Yaskawa INFORM job: KRIS3(-160_-90)54.JBI

/JOB
//NAME KRIS3(-160_-90)54
//POS
///NPOS 270,270,270,20,0,0
///TOOL 0
///POSTYPE PULSE
///PULSE
C00000=36470,-76528,-106815,-19279,71473,-77234
C00001=136908,-99459,-124829,-20670,71348,-76391
C00002=134470,-76528,-106815,-19279,71473,-77234
C00003=159578,-94739,-111578,-14965,102577,-71346
C00004=157566,-87256,-71357,-3912,80960,-68626
C00005=176880,-68125,-57902,-5422,83635,-62119
C00006=177907,-68461,-55745,-5507,82211,-61705
C00007=177907,-68063,-54493,-5513,81648,-61681
C00008=177907,-68139,-54730,-5512,81754,-61686
C00009=178677,-69433,-55362,-5571,81531,-61412
C00010=178017,-68613,-55721,-5516,82126,-61665
C00011=169648,-85474,-89038,-4887,93378,-64966
C00012=163611,-44630,-68122,-4506,101126,-67267
C00013=165231,-48362,-64740,-4579,97228,-66587
C00014=165334,-48746,-64513,-4584,96897,-66540
C00015=165334,-48893,-63576,-4578,96247,-66515
C00016=165334,-48879,-63681,-4579,96319,-66517
C00017=165646,-49837,-64080,-4605,96090,-66402
C00018=165334,-48746,-64513,-4584,96897,-66540
C00019=140979,-108094,-110643,-2385,93763,-74547
C00020=140979,-108094,-110643,-2385,93763,-74547
C00021=140979,-108094,-110643,-2385,93763,-74547
C00022=140979,-108094,-110643,-2385,93763,-74547
C00023=140979,-108246,-109289,-2383,92853,-74530
C00024=140979,-108231,-109453,-2383,92961,-74533
C00025=141280,-110659,-110301,-2409,92244,-74420
C00026=140979,-108094,-110643,-2385,93763,-74547
C00027=156700,-55897,-85418,8720,99373,-67438
C00028=156898,-58036,-83987,8629,97394,-67513
C00029=156898,-58722,-82817,8603,96332,-67586
C00030=156898,-58622,-82997,8608,96491,-67574
C00031=157341,-60416,-83948,8523,96115,-67457
C00032=156898,-58036,-83987,8629,97394,-67513
C00033=161369,-86849,-99090,-4273,98390,-67906
C00034=167909,-84037,-82934,3708,84523,-64877
C00035=168571,-85124,-82512,3609,83677,-64677
C00036=168571,-84898,-80901,3613,82804,-64704
C00037=168571,-84936,-81149,3613,82937,-64700
C00038=169203,-86467,-81802,3516,82525,-64499
C00039=168571,-85124,-82512,3609,83677,-64677
C00040=165600,-121955,-98284,4061,74695,-65975
C00041=174461,-109455,-70225,9835,59183,-64105
C00042=175080,-109402,-69148,9749,58483,-63930
C00043=175080,-108469,-67668,9792,58058,-63969
C00044=175080,-108628,-67921,9785,58130,-63962
C00045=176152,-109889,-68298,9565,57596,-63593
C00046=175080,-109402,-69148,9749,58483,-63930
C00047=145436,-132582,-96247,390,75065,-72870
C00048=145436,-132678,-96385,390,75101,-72870
C00049=145436,-153478,-122593,390,33069,-72870
C00050=145436,-153478,-122593,390,33069,-72870
C00051=145875,-137224,-99164,151,44123,-76557
C00052=145875,-137224,-99164,-3186,26783,-75636
C00053=145875,-137224,-99164,-3186,26783,-75636
C00054=126920,-141995,-100488,14842,27437,-88451
C00055=126921,-139435,-97257,15195,26791,-88624
C00056=126921,-140260,-98306,15082,27005,-88567
C00057=126657,-136107,-97292,14665,28515,-88375
C00058=126920,-141995,-100488,14842,27437,-88451
C00059=153689,-122615,-92358,7246,28662,-82796
C00060=153689,-122359,-91923,7277,28527,-82812
C00061=153689,-121251,-90046,7417,27945,-82882
C00062=153689,-121596,-90629,7373,28125,-82859
C00063=152562,-118169,-89603,8504,29355,-83484
C00064=153689,-122359,-91923,7277,28527,-82812
C00065=153734,-144670,-102026,-12528,26386,-79802
C00066=148920,-141423,-91163,-14854,15551,-80235
C00067=148967,-137496,-86916,-15534,14983,-79917
C00068=147891,-134819,-86332,-12174,15793,-81580
C00069=147123,-134668,-89168,-6588,20492,-83847
C00070=147184,-133728,-87772,-6813,20125,-83735
C00071=149705,-139389,-87494,-17948,14535,-78726
C00072=140769,-160579,-91179,-72763,19950,-46602
C00073=129302,-154781,-89703,-59410,13959,-54584
C00074=128993,-152913,-89439,-56337,14227,-56040
C00075=129214,-154274,-89633,-58559,14027,-54988
C00076=129214,-151990,-87339,-59384,13900,-54610
C00077=129539,-156129,-91089,-59119,14177,-54682
C00078=130002,-156587,-91482,-58522,14566,-54861
C00079=131612,-152018,-92345,-56188,18115,-55777
C00080=137260,-138866,-133764,-10166,31487,-76482
C00081=55962,-149633,-123442,-11923,14089,-75671
C00082=31464,-162597,-133764,-10166,12061,-76482
C00083=-11401,-148032,-125425,-11667,35640,-75771
C00084=-126225,-114648,-117375,-36487,17100,-65054
C00085=-160935,-140983,-109640,-13468,75088,-74332
C00086=-169853,-118963,-84593,-12681,69660,86771
C00087=-166041,-110678,-74459,-13320,68331,88303
C00088=-166223,-108797,-70951,-13405,67140,88373
C00089=-166223,-107663,-69097,-13458,66595,88438
C00090=-166223,-107867,-69431,-13449,66693,88427
C00091=-167322,-109580,-69957,-13369,65975,88109
C00092=-166243,-109210,-71582,-13386,67309,88347
C00093=-169217,-106350,-70409,-12947,67561,87233
C00094=-169217,-106256,-70250,-12951,67512,87238
C00095=-169217,-105112,-68312,-13006,66921,87306
C00096=-169217,-105283,-68599,-12998,67008,87297
C00097=-170397,-106999,-69102,-12897,66265,86949
C00098=-167930,-107758,-71144,-13135,67501,87709
C00099=-168330,-125239,-100831,-12460,76505,86600
C00100=-155830,-85289,-85709,-13656,89459,89593
C00101=-155617,-85922,-82565,-13677,87294,89905
C00102=-155617,-85683,-81004,-13681,86480,89993
C00103=-155617,-85728,-81276,-13680,86620,89979
C00104=-156391,-88450,-82422,-13606,85816,89798
C00105=-155763,-86416,-82528,-13661,87001,89886
C00106=-155923,-87175,-84120,-13644,87549,89771
C00107=-155609,-85916,-82709,-13676,87386,89897
C00108=-155609,-85729,-81437,-13679,86718,89971
C00109=-155609,-85763,-81652,-13678,86829,89960
C00110=-156185,-87803,-82513,-13623,86229,89826
C00111=-155614,-85958,-82864,-13674,87458,89888
C00112=-155923,-85281,-100905,-13881,98543,88548
C00113=-155518,-83496,-100141,-13947,99043,88626
C00114=-155147,-83263,-96119,-13888,96814,89004
C00115=-155147,-83507,-95337,-13865,96223,89071
C00116=-155147,-83457,-95507,-13869,96351,89056
C00117=-155768,-86094,-96638,-13778,95608,88929
C00118=-155255,-83510,-96958,-13888,97175,88925
C00119=-154682,-87233,-101845,693,104782,88208
C00120=-154005,-85079,-98247,676,103668,88429
C00121=-154005,-85354,-97445,675,103031,88426
C00122=-154005,-85287,-97652,675,103193,88426
C00123=-154486,-87439,-98578,683,102661,88260
C00124=-154216,-85718,-99521,682,104126,88361
C00125=-156826,-87943,-103938,737,105722,87490
C00126=-169505,-149944,-134809,912,70958,83129
C00127=-207316,-122712,-123448,7636,86368,80631
C00128=-224855,-108358,-71229,12006,64036,72649
C00129=-217077,-74631,-23766,41947,48629,49537
C00130=-218892,-67424,-12026,68960,50607,41965
C00131=-212692,-64398,-6060,71724,46143,41638
C00132=-212692,-63310,-4348,72177,45977,41343
C00133=-212692,-64398,-6060,71724,46143,41638
C00134=-210575,-63691,-5764,71905,44943,42037
C00135=-212692,-64398,-6060,71724,46143,41638
C00136=-222676,-51835,-4012,66283,54122,43011
C00137=-220683,-43055,3882,66739,52777,43150
C00138=-220683,-41728,6197,67257,52470,42760
C00139=-220683,-43055,3882,66739,52777,43150
C00140=-218176,-42178,4378,66898,51329,43628
C00141=-220683,-43055,3882,66739,52777,43150
C00142=-234013,-57846,-7460,65247,60464,40769
C00143=-233739,-55371,-8506,61318,66043,45868
C00144=-224021,-72963,-6178,68579,55797,42417
C00145=-222956,-69762,-1623,69618,54766,41957
C00146=-220957,-69447,-1516,70121,53696,42256
C00147=-222193,-69648,-1584,69812,54356,42072
C00148=-222502,-68090,774,70157,54288,41693
C00149=-222193,-69648,-1584,69812,54356,42072
C00150=-225636,-56152,5458,67261,57288,42948
C00151=-149006,-93113,-100988,5480,101691,74295
C00152=-149599,-96300,-103483,5484,101628,74092
C00153=-219127,-73013,-224,68618,57817,46460
C00154=-228607,-72912,-7621,63442,64869,47367
C00155=-220423,-75882,-15995,70402,50905,40654
C00156=-212092,-63463,-4317,72649,45688,41298
C00157=-163022,-96735,-99152,-22140,103253,76925
C00158=-162158,-93804,-96763,-22109,103515,77196
C00159=-220673,-36477,9481,67037,52832,43066
C00160=-225006,-42245,766,65045,56479,43585
C00161=-234485,-59648,-18556,62655,63569,43382
C00162=-203757,-97365,-58564,4219,60682,62576
C00163=-234472,-129171,-97928,9356,71113,51987
C00164=-234472,-150736,-135181,8964,82814,52858
C00165=-234472,-150736,-135181,8964,82814,52858
C00166=-215909,-75798,-109600,6127,103741,60188
C00167=-142211,-189130,-127292,69248,52498,52988
C00168=-118502,-172484,-110233,52609,25212,65150
C00169=-171509,-133648,-100111,8061,78079,67623
C00170=-179980,-112353,-73580,8533,73608,64392
C00171=-172896,-96696,-66298,2439,82915,67706
C00172=-163006,-94576,-83573,-21494,95359,78388
C00173=-162142,-91714,-81191,-21448,95589,78662
C00174=-161445,-106166,-69505,2991,79646,71488
C00175=-161519,-107811,-73451,2977,81228,71500
C00176=-162580,-105162,-72246,-8409,75537,72147
C00177=-166515,-102401,-68173,-8273,74056,70883
C00178=-163006,-94576,-83573,-21494,95359,78388
C00179=-162142,-91714,-81191,-21448,95589,78662
C00180=-175761,-93408,-64742,-7691,75635,67570
C00181=-169252,-115124,-101169,-7872,87423,69075
C00182=-154261,-79873,-81468,-8571,94879,73696
C00183=-155062,-80931,-79256,-8513,92911,73559
C00184=-163006,-94576,-83573,-21494,95359,78388
C00185=-162142,-91714,-81191,-21448,95589,78662
C00186=-163211,-72770,-75533,-8210,93956,70713
C00187=-163718,-69809,-76291,-8220,95872,70416
C00188=-152145,-81088,-82167,-2065,97703,74759
C00189=-153291,-82185,-80570,-2065,96129,74395
C00190=-163006,-94576,-83573,-21494,95359,78388
C00191=-162142,-91714,-81191,-21448,95589,78662
C00192=-143402,-88471,-83234,-1964,94787,77778
C00193=-144574,-84995,-103251,-2104,108854,77145
C00194=-151765,-102418,-106955,5657,95758,75438
C00195=-150608,-101637,-104194,5548,94387,75768
C00196=-163006,-94576,-83573,-21494,95359,78388
C00197=-162142,-91714,-81191,-21448,95589,78662
C00198=-139211,-109713,-107103,4584,91330,79466
C00199=-143989,-108966,-109417,5008,93413,77941
C00200=-143223,-109509,-108756,-8615,88663,77081
C00201=-143797,-107565,-105457,-8538,87583,76960
C00202=-163006,-94576,-83573,-21494,95359,78388
C00203=-162142,-91714,-81191,-21448,95589,78662
C00204=-154250,-98677,-102309,-7016,89198,73353
C00205=-144143,-146387,-128453,-8544,81812,77235
C00206=-130399,-165491,-128261,582,73715,81342
C00207=-149731,-158641,-113843,-14975,70738,-69794
C00208=-149731,-158641,-113843,-14975,70738,-69794
C00209=-126225,-114648,-117375,-36487,17100,-65054
C00210=-118781,-153853,-134406,-32592,23357,-65054
C00211=-12470,-167083,-125425,-11667,16324,-75771
C00212=137258,-84249,-120477,-10166,64820,-76482
C00213=160540,-100857,-113063,-23155,68829,-67581
C00214=182830,-114405,-112845,-16003,91175,-61677
C00215=183790,-123536,-112279,-16086,86512,-60735
C00216=173929,-95305,-100930,-8088,100256,-64859
C00217=158743,-95268,-103371,-5812,102972,-69826
C00218=157888,-92366,-100981,-5813,102933,-70115
C00219=164971,-109182,-106036,-7793,95435,-67600
C00220=164197,-113877,-111682,-7800,96401,-67923
C00221=173870,-143306,-120553,-7913,87764,-64082
C00222=171816,-118751,-98057,-3590,91441,-64891
C00223=176035,-116344,-93182,-3358,89860,-63416
C00224=158755,-94787,-86481,976,103949,-69303
C00225=157900,-91912,-84097,841,103969,-69603
C00226=165474,-127613,-96498,-3911,85645,-66872
C00227=163756,-130674,-100363,-3993,86365,-67475
C00228=177254,-154866,-106204,-3341,78153,-62695
C00229=194740,-128784,-79093,-2289,75465,-56815
C00230=199705,-123555,-74669,-1955,75552,-55172
C00231=158782,-86330,-62292,-2348,97119,-70521
C00232=157926,-83586,-59872,-2521,97014,-70811
C00233=188878,-135549,-77220,-2730,70669,-58654
C00234=186334,-138981,-80518,-2891,70851,-59497
C00235=202790,-114657,-73561,7469,64730,-55511
C00236=205310,-109506,-69417,7096,64604,-54603
C00237=158743,-95268,-103371,-5812,102972,-69826
C00238=157888,-92366,-100981,-5813,102933,-70115
C00239=208506,-101173,-65845,8459,63334,-53705
C00240=188075,-151957,-103997,12598,63075,-61358
C00241=175676,-115929,-94468,13375,77380,-64283
C00242=179228,-108031,-88427,12897,77138,-63049
C00243=158755,-94787,-86481,976,103949,-69303
C00244=157900,-91912,-84097,841,103969,-69603
C00245=187549,-93923,-83081,11553,79750,-59861
C00246=178297,-108275,-107099,12771,88378,-62209
C00247=165278,-79866,-95804,14582,97947,-65562
C00248=167332,-81697,-93226,14245,95145,-65199
C00249=158782,-86330,-62292,-2348,97119,-70521
C00250=157926,-83586,-59872,-2521,97014,-70811
C00251=172083,-74876,-89232,15991,93470,-63478
C00252=166883,-83368,-97274,16810,95013,-65031
C00253=148381,-154133,-120540,18986,77988,-74048
C00254=148381,-154133,-120540,18986,29025,-74048
C00255=148381,-154133,-120540,18986,29025,-74048
C00256=148381,-154133,-120540,18986,29025,-74048
C00257=148381,-154133,-120540,635,27393,-68347
C00258=131809,-160671,-109428,31686,20564,-84507
C00259=131822,-150122,-103532,29341,22114,-83385
C00260=161827,-137088,-100610,-19196,25445,-57865
C00261=160079,-162229,-113551,-20584,20355,-57319
C00262=127848,-170739,-113822,-25929,20694,-59837
C00263=98584,-145628,-105124,27441,32859,-85558
C00264=101235,-136742,-99408,24366,32991,-83733
C00265=148832,-132035,-98353,-25409,35327,-54782
C00266=162526,-150393,-107796,-38053,37342,-46820
C00267=161637,-148332,-107324,-36893,37578,-47548
C00268=136473,-81821,-106853,-20577,68974,-75046
C00269=36470,-76528,-106815,-19279,71473,-77234
BC00000=293716,514317,1072451
BC00001=351926,331601,1072451
BC00002=351926,292903,1072451
BC00003=351926,213013,1072451
BC00004=381341,211891,1072451
BC00005=381341,211891,1072451
BC00006=381341,211891,1072451
BC00007=381341,211891,1072451
BC00008=381341,211891,1072451
BC00009=381341,211891,1072451
BC00010=381341,211891,1072451
BC00011=381341,211891,1072448
BC00012=381341,211891,1072448
BC00013=381341,211891,1072448
BC00014=381341,211891,1072448
BC00015=381341,211891,1072448
BC00016=381341,211891,1072448
BC00017=381341,211891,1072448
BC00018=381341,211891,1072448
BC00019=327940,182383,1072451
BC00020=327940,158933,1072451
BC00021=323570,159157,1054517
BC00022=322810,158773,1051038
BC00023=322810,158773,1051038
BC00024=322810,158773,1051038
BC00025=322810,158773,1051038
BC00026=322810,158773,1051038
BC00027=324758,182517,1072451
BC00028=324758,182517,1072451
BC00029=324758,182517,1072451
BC00030=324758,182517,1072451
BC00031=324758,182517,1072451
BC00032=324758,182517,1072451
BC00033=323103,182517,1072451
BC00034=323103,182517,1072451
BC00035=323103,182517,1072451
BC00036=323103,182517,1072451
BC00037=323103,182517,1072451
BC00038=323103,182517,1072451
BC00039=323103,182517,1072451
BC00040=323103,182517,1072451
BC00041=323103,182517,1072451
BC00042=323103,182517,1072451
BC00043=323103,182517,1072451
BC00044=323103,182517,1072451
BC00045=323103,182517,1072451
BC00046=323103,182517,1072451
BC00047=332426,182517,1072451
BC00048=332426,182517,1072451
BC00049=332426,227917,1072451
BC00050=367924,391941,1072451
BC00051=367924,391941,1072451
BC00052=323298,308265,712615
BC00053=297724,284937,708891
BC00054=297724,284937,708891
BC00055=297724,284937,708889
BC00056=297724,284937,708889
BC00057=297724,284937,708889
BC00058=297724,284937,708891
BC00059=297724,284937,708891
BC00060=297724,284937,708891
BC00061=297724,284937,708891
BC00062=297724,284937,708891
BC00063=297724,284937,708891
BC00064=297724,284937,708891
BC00065=325419,295206,714526
BC00066=325419,295206,704236
BC00067=325419,295206,704234
BC00068=325419,295206,704234
BC00069=325419,295206,704234
BC00070=325419,295206,704234
BC00071=325419,295206,704234
BC00072=319446,285786,704234
BC00073=319446,285786,704234
BC00074=319446,285786,704234
BC00075=319446,285786,704234
BC00076=319446,285786,704234
BC00077=319446,285786,704234
BC00078=306058,333731,968548
BC00079=310610,415570,1064706
BC00080=352207,264891,1072451
BC00081=372153,109357,1072451
BC00082=378164,62489,1072451
BC00083=396581,158595,1072451
BC00084=311023,50823,1072451
BC00085=339144,73580,1072451
BC00086=339157,74032,1072451
BC00087=339157,74032,1072451
BC00088=339157,74032,1072451
BC00089=339157,74032,1072451
BC00090=339157,74032,1072451
BC00091=339157,74032,1072451
BC00092=339157,74032,1072451
BC00093=372221,74032,1072451
BC00094=372221,74032,1072451
BC00095=372221,74032,1072451
BC00096=372221,74032,1072451
BC00097=372221,74032,1072451
BC00098=372221,74032,1072451
BC00099=372221,74032,1072451
BC00100=372221,74032,1072451
BC00101=372221,74032,1072451
BC00102=372221,74032,1072451
BC00103=372221,74032,1072451
BC00104=372221,74032,1072451
BC00105=372221,74032,1072451
BC00106=338445,74032,1072451
BC00107=338445,73232,1069168
BC00108=338445,73232,1069168
BC00109=338445,73232,1069168
BC00110=338445,73232,1069168
BC00111=338445,73232,1069168
BC00112=338445,73232,1071030
BC00113=338445,99622,1071030
BC00114=338445,99622,1071030
BC00115=338445,99622,1071030
BC00116=338445,99622,1071030
BC00117=338445,99622,1071030
BC00118=338445,99622,1071030
BC00119=338445,99622,1071030
BC00120=338445,99622,1071030
BC00121=338445,99622,1071030
BC00122=338445,99622,1071030
BC00123=338445,99622,1071030
BC00124=338445,99622,1071030
BC00125=338445,99622,1071030
BC00126=338445,99622,1071030
BC00127=395065,437,1069903
BC00128=395065,437,1069903
BC00129=395065,437,1069903
BC00130=395065,437,1069903
BC00131=395065,437,1069903
BC00132=395065,437,1069903
BC00133=395065,437,1069903
BC00134=395065,437,1069903
BC00135=395065,437,1069903
BC00136=395065,437,1069903
BC00137=395065,437,1069903
BC00138=395065,437,1069903
BC00139=395065,437,1069903
BC00140=395065,437,1069903
BC00141=395065,437,1069903
BC00142=395065,437,1069903
BC00143=395064,1123,1069901
BC00144=395064,1123,1069901
BC00145=395064,1123,1069901
BC00146=395064,1123,1069901
BC00147=395064,1123,1069901
BC00148=395064,1123,1069901
BC00149=395064,1123,1069901
BC00150=395064,1123,1069901
BC00151=347303,98646,1072451
BC00152=347303,98646,1072451
BC00153=395064,1123,1069901
BC00154=395064,1123,1069901
BC00155=395064,1123,1069901
BC00156=395064,1123,1069901
BC00157=320927,137430,1072451
BC00158=320927,137430,1072451
BC00159=395064,1123,1069901
BC00160=395064,1123,1069901
BC00161=395064,1123,1069901
BC00162=395064,1123,1069901
BC00163=395064,22229,1069901
BC00164=395064,22229,1069901
BC00165=395064,111405,1069901
BC00166=395064,111405,1069901
BC00167=307195,19114,1039924
BC00168=312628,21569,1045452
BC00169=339157,74031,1072445
BC00170=339157,74031,1072445
BC00171=339157,74031,1072445
BC00172=320853,110629,1072451
BC00173=320853,110629,1072451
BC00174=339157,74031,1072445
BC00175=339157,74031,1072445
BC00176=339157,74031,1072445
BC00177=339157,74031,1072445
BC00178=320853,110629,1072451
BC00179=320853,110629,1072451
BC00180=339157,74031,1072445
BC00181=339157,74031,1072445
BC00182=339157,74031,1072445
BC00183=339157,74031,1072445
BC00184=320853,110629,1072451
BC00185=320853,110629,1072451
BC00186=339157,74031,1072445
BC00187=339157,74031,1072445
BC00188=339157,74031,1072445
BC00189=339157,74031,1072445
BC00190=320853,110629,1072451
BC00191=320853,110629,1072451
BC00192=339157,74031,1072445
BC00193=339157,74031,1072445
BC00194=321867,96463,1067741
BC00195=321867,96463,1067741
BC00196=320853,110629,1072451
BC00197=320853,110629,1072451
BC00198=321867,96463,1067741
BC00199=321867,96463,1067741
BC00200=321867,96463,1067741
BC00201=321867,96463,1067741
BC00202=320853,110629,1072451
BC00203=320853,110629,1072451
BC00204=321867,96463,1067741
BC00205=321867,96463,1067741
BC00206=331832,83535,1070452
BC00207=339144,73580,1072451
BC00208=339144,73580,1072451
BC00209=311023,50823,1072451
BC00210=311023,50823,1072451
BC00211=396581,158595,1072451
BC00212=352208,264890,1072451
BC00213=380287,222292,1072451
BC00214=345793,144315,1072448
BC00215=345793,144315,1072448
BC00216=345793,144315,1072448
BC00217=363046,147874,1072451
BC00218=363046,147874,1072451
BC00219=345793,144315,1072448
BC00220=346013,144317,1072448
BC00221=346013,144317,1072448
BC00222=336959,144429,1072450
BC00223=336960,144428,1072447
BC00224=363165,149824,1072451
BC00225=363165,149824,1072451
BC00226=336960,144428,1072447
BC00227=336960,144428,1072447
BC00228=336960,144428,1072447
BC00229=336960,144428,1072447
BC00230=336960,144428,1072447
BC00231=353911,176435,1072451
BC00232=353911,176435,1072451
BC00233=336960,144428,1072447
BC00234=336960,144428,1072447
BC00235=336960,144428,1072447
BC00236=336960,144428,1072447
BC00237=363046,147874,1072451
BC00238=363046,147874,1072451
BC00239=336960,144428,1072447
BC00240=336960,144428,1072447
BC00241=336960,144428,1072447
BC00242=336960,144428,1072447
BC00243=363165,149824,1072451
BC00244=363165,149824,1072451
BC00245=336960,144428,1072447
BC00246=336960,144428,1072447
BC00247=336960,144428,1072447
BC00248=336960,144428,1072447
BC00249=353911,176435,1072451
BC00250=353911,176435,1072451
BC00251=336960,144428,1072447
BC00252=336960,144428,1072447
BC00253=336960,144428,1072447
BC00254=376956,227130,1072447
BC00255=384452,390236,1072447
BC00256=384452,390236,786592
BC00257=345962,304340,657091
BC00258=316411,279825,657091
BC00259=316411,279825,657091
BC00260=299501,279825,657091
BC00261=316411,279825,657091
BC00262=329749,298472,657091
BC00263=315017,300783,657091
BC00264=315017,300783,657091
BC00265=312927,300783,657091
BC00266=315017,300783,657091
BC00267=315017,430587,912822
BC00268=349205,500385,1060684
BC00269=293716,514317,1072451
EC00000=1418945,372643
EC00001=1418945,372643
EC00002=1418945,372643
EC00003=1418945,372643
EC00004=1418945,372643
EC00005=1418945,372643
EC00006=1418945,372643
EC00007=1418945,372643
EC00008=1418945,372643
EC00009=1418945,372643
EC00010=1418945,372643
EC00011=1418944,372643
EC00012=1418944,372643
EC00013=1418944,372643
EC00014=1418944,372643
EC00015=1418944,372643
EC00016=1418944,372643
EC00017=1418944,372643
EC00018=1418944,372643
EC00019=1418945,372643
EC00020=1418945,372643
EC00021=1418945,372643
EC00022=1418945,372643
EC00023=1418945,372643
EC00024=1418945,372643
EC00025=1418945,372643
EC00026=1418945,372643
EC00027=1418945,372643
EC00028=1418945,372643
EC00029=1418945,372643
EC00030=1418945,372643
EC00031=1418945,372643
EC00032=1418945,372643
EC00033=1418945,372643
EC00034=1418945,372643
EC00035=1418945,372643
EC00036=1418945,372643
EC00037=1418945,372643
EC00038=1418945,372643
EC00039=1418945,372643
EC00040=1418945,372643
EC00041=1418945,372643
EC00042=1418945,372643
EC00043=1418945,372643
EC00044=1418945,372643
EC00045=1418945,372643
EC00046=1418945,372643
EC00047=1418945,372643
EC00048=1418945,372643
EC00049=1418945,372643
EC00050=1418945,372643
EC00051=1418945,372643
EC00052=1418945,372643
EC00053=1418945,372643
EC00054=1418945,372643
EC00055=1418944,372643
EC00056=1418944,372643
EC00057=1418944,372643
EC00058=1418945,372643
EC00059=1418945,372643
EC00060=1418945,372643
EC00061=1418945,372643
EC00062=1418945,372643
EC00063=1418945,372643
EC00064=1418945,372643
EC00065=1418945,372643
EC00066=1418945,372643
EC00067=1418945,372643
EC00068=1418945,372643
EC00069=1418945,372643
EC00070=1418945,372643
EC00071=1418945,372643
EC00072=1418945,372643
EC00073=1418945,372643
EC00074=1418945,372643
EC00075=1418945,372643
EC00076=1418945,372643
EC00077=1418945,372643
EC00078=1418945,372643
EC00079=1418945,372643
EC00080=1418945,372643
EC00081=1418945,372643
EC00082=1418945,372643
EC00083=1595090,-179995
EC00084=1773681,-740307
EC00085=1773681,-740307
EC00086=1773681,-740307
EC00087=1773681,-740307
EC00088=1773681,-740307
EC00089=1773681,-740307
EC00090=1773681,-740307
EC00091=1773681,-740307
EC00092=1773681,-740307
EC00093=1773681,-740307
EC00094=1773681,-740307
EC00095=1773681,-740307
EC00096=1773681,-740307
EC00097=1773681,-740307
EC00098=1773681,-740307
EC00099=1773681,-740307
EC00100=1773681,-740307
EC00101=1773681,-740307
EC00102=1773681,-740307
EC00103=1773681,-740307
EC00104=1773681,-740307
EC00105=1773681,-740307
EC00106=1773681,-740307
EC00107=1773681,-740307
EC00108=1773681,-740307
EC00109=1773681,-740307
EC00110=1773681,-740307
EC00111=1773681,-740307
EC00112=1773681,-740307
EC00113=1773681,-740307
EC00114=1773681,-740307
EC00115=1773681,-740307
EC00116=1773681,-740307
EC00117=1773681,-740307
EC00118=1773681,-740307
EC00119=1773681,-740307
EC00120=1773681,-740307
EC00121=1773681,-740307
EC00122=1773681,-740307
EC00123=1773681,-740307
EC00124=1773681,-740307
EC00125=1773681,-740307
EC00126=1773681,-740307
EC00127=1773681,-740307
EC00128=1773681,-740307
EC00129=1773681,-740307
EC00130=1773681,-740307
EC00131=1773681,-740307
EC00132=1773681,-740307
EC00133=1773681,-740307
EC00134=1773681,-740307
EC00135=1773681,-740307
EC00136=1773681,-740307
EC00137=1773681,-740307
EC00138=1773681,-740307
EC00139=1773681,-740307
EC00140=1773681,-740307
EC00141=1773681,-740307
EC00142=1773681,-740307
EC00143=1773685,-740307
EC00144=1773685,-740307
EC00145=1773685,-740307
EC00146=1773685,-740307
EC00147=1773685,-740307
EC00148=1773685,-740307
EC00149=1773685,-740307
EC00150=1773685,-740307
EC00151=1773681,-740307
EC00152=1773681,-740307
EC00153=1773685,-740307
EC00154=1773685,-740307
EC00155=1773685,-740307
EC00156=1773685,-740307
EC00157=1773681,-740307
EC00158=1773681,-740307
EC00159=1773685,-740307
EC00160=1773685,-740307
EC00161=1773685,-740307
EC00162=1773685,-740307
EC00163=1773685,-740307
EC00164=1773685,-740307
EC00165=1773685,-740307
EC00166=1773685,-740307
EC00167=1773681,-740307
EC00168=1773681,-740307
EC00169=1773683,-740305
EC00170=1773683,-740305
EC00171=1773683,-740305
EC00172=1773681,-740307
EC00173=1773681,-740307
EC00174=1773683,-740305
EC00175=1773683,-740305
EC00176=1773683,-740305
EC00177=1773683,-740305
EC00178=1773681,-740307
EC00179=1773681,-740307
EC00180=1773683,-740305
EC00181=1773683,-740305
EC00182=1773683,-740305
EC00183=1773683,-740305
EC00184=1773681,-740307
EC00185=1773681,-740307
EC00186=1773683,-740305
EC00187=1773683,-740305
EC00188=1773683,-740305
EC00189=1773683,-740305
EC00190=1773681,-740307
EC00191=1773681,-740307
EC00192=1773683,-740305
EC00193=1773683,-740305
EC00194=1773683,-740305
EC00195=1773683,-740305
EC00196=1773681,-740307
EC00197=1773681,-740307
EC00198=1773683,-740305
EC00199=1773683,-740305
EC00200=1773683,-740305
EC00201=1773683,-740305
EC00202=1773681,-740307
EC00203=1773681,-740307
EC00204=1773683,-740305
EC00205=1773683,-740305
EC00206=1773683,-740305
EC00207=1773681,-740307
EC00208=1773681,-740307
EC00209=1773681,-740307
EC00210=1773681,-740307
EC00211=1595090,-179995
EC00212=1418947,372636
EC00213=1418945,372643
EC00214=1418944,372643
EC00215=1418944,372643
EC00216=1418944,372643
EC00217=1418945,372643
EC00218=1418945,372643
EC00219=1418944,372643
EC00220=1418944,372643
EC00221=1418944,372643
EC00222=1418945,372643
EC00223=1418944,372643
EC00224=1418945,372643
EC00225=1418945,372643
EC00226=1418944,372643
EC00227=1418944,372643
EC00228=1418944,372643
EC00229=1418944,372643
EC00230=1418944,372643
EC00231=1418945,372643
EC00232=1418945,372643
EC00233=1418944,372643
EC00234=1418944,372643
EC00235=1418944,372643
EC00236=1418944,372643
EC00237=1418945,372643
EC00238=1418945,372643
EC00239=1418944,372643
EC00240=1418944,372643
EC00241=1418944,372643
EC00242=1418944,372643
EC00243=1418945,372643
EC00244=1418945,372643
EC00245=1418944,372643
EC00246=1418944,372643
EC00247=1418944,372643
EC00248=1418944,372643
EC00249=1418945,372643
EC00250=1418945,372643
EC00251=1418944,372643
EC00252=1418944,372643
EC00253=1418944,372643
EC00254=1418944,372643
EC00255=1418944,372643
EC00256=1418944,372643
EC00257=1418944,372643
EC00258=1418944,372643
EC00259=1418944,372643
EC00260=1418944,372643
EC00261=1418944,372643
EC00262=1418944,372643
EC00263=1418944,372643
EC00264=1418944,372643
EC00265=1418944,372643
EC00266=1418944,372643
EC00267=1418944,372643
EC00268=1418945,372643
EC00269=1418945,372643
///POSTYPE BASE
///RECTAN
///RCONF 0,0,0,0,1,0,0,0,0,0,0,0,0,0,0,0,0,0,0,0,0,0,0,0
P00006=2.006,1.622,-0.565,0.0000,0.0000,0.0000
P00021=0.073,2.058,-0.109,0.0000,0.0000,0.0000
P00022=2.006,1.622,-0.565,0.0000,0.0000,0.0000
///RCONF 0,0,0,0,0,0,0,0,0,0,0,0,0,0,0,0,0,0,0,0,0,0,0,0
P00023=-2.957,-4.083,2.762,0.0000,0.0000,0.0000
P00024=-1.466,-0.226,-0.419,0.0000,0.0000,0.0000
P00025=3.643,0.007,-2.585,0.0000,0.0000,0.0000
P00026=2.644,0.055,-2.583,0.0000,0.0000,0.0000
P00027=2.278,0.099,-4.210,0.0000,0.0000,0.0000
P00028=-1.778,-0.182,-2.050,0.0000,0.0000,0.0000
P00029=1.749,4.006,-0.261,0.0000,0.0000,0.0000
P00030=-0.014,-0.768,0.131,0.0000,0.0000,0.0000
P00031=-0.170,0.039,-0.647,0.0000,0.0000,0.0000
P00032=-0.423,0.157,3.222,0.0000,0.0000,0.0000
P00033=0.854,-1.099,3.047,0.0000,0.0000,0.0000
///RCONF 0,0,0,0,1,0,0,0,0,0,0,0,0,0,0,0,0,0,0,0,0,0,0,0
P00034=-8.151,9.743,-4.393,0.0000,0.0000,0.0000
///RCONF 0,0,0,0,0,0,0,0,0,0,0,0,0,0,0,0,0,0,0,0,0,0,0,0
P00035=0.390,-0.027,1.040,0.0000,0.0000,0.0000
P00036=-2.434,0.084,0.197,0.0000,0.0000,0.0000
P00037=-1.075,5.090,-3.949,0.0000,0.0000,0.0000
P00038=0.174,-1.527,-10.860,0.0000,0.0000,0.0000
P00039=-0.109,1.838,-0.266,0.0000,0.0000,0.0000
//INST
///DATE 2024/11/25 20:44
///ATTR SC,RW
///GROUP1 RB1,BS1
///GROUP2 ST1
NOP
MOVJ C00000 BC00000 VJ=100.00  +MOVJ EC00000 VJ=100.00
'MUZYLO 260124 START
MOVJ C00001 BC00001 VJ=100.00  +MOVJ EC00001 VJ=100.00
MOVJ C00002 BC00002 VJ=100.00  +MOVJ EC00002 VJ=100.00
MOVJ C00003 BC00003 VJ=100.00  +MOVJ EC00003 VJ=100.00
'Path S1422
SFTOF3D
MOVJ C00004 BC00004 VJ=100.00  +MOVJ EC00004 VJ=100.00
MOVL C00005 BC00005 V=400.0  +MOVJ EC00005 VJ=100.00
SMOVL C00006 BC00006 V=100.0  +MOVJ EC00006
SREFP 3 C00007 BC00007  +REFP EC00007
CALL JOB:SEARCH-R1-S13D
SET P021 P006
SFTON3D P021
SMOVL C00008 BC00008 V=100.0  +MOVJ EC00008
SREFP 3 C00009 BC00009  +REFP EC00009
CALL JOB:SEARCH-R1-S13D
SET P021 P006
SFTON3D P021
SMOVL C00010 BC00010 V=100.0  +MOVJ EC00010
MOVL C00011 BC00011 V=400.0  +MOVJ EC00011 VJ=100.00
MOVL C00012 BC00012 V=1000.0  +MOVJ EC00012 VJ=100.00
MOVJ C00013 BC00013 VJ=100.00  +MOVJ EC00013 VJ=100.00
'Path S1423
SFTOF3D
SMOVL C00014 BC00014 V=100.0  +MOVJ EC00014
SREFP 3 C00015 BC00015  +REFP EC00015
CALL JOB:SEARCH-R1-S13D
SET P022 P006
SFTON3D P022
SMOVL C00016 BC00016 V=100.0  +MOVJ EC00016
SREFP 3 C00017 BC00017  +REFP EC00017
CALL JOB:SEARCH-R1-S13D
SET P022 P006
SFTON3D P022
SMOVL C00018 BC00018 V=100.0  +MOVJ EC00018
MOVL C00019 BC00019 V=400.0  +MOVJ EC00019 VJ=100.00
MOVL C00020 BC00020 V=1000.0  +MOVJ EC00020 VJ=100.00
MOVJ C00021 BC00021 VJ=100.00  +MOVJ EC00021 VJ=100.00
'Path S1424
SFTOF3D
SMOVL C00022 BC00022 V=100.0  +MOVJ EC00022
SREFP 3 C00023 BC00023  +REFP EC00023
CALL JOB:SEARCH-R1-S13D
SET P023 P006
SFTON3D P023
SMOVL C00024 BC00024 V=100.0  +MOVJ EC00024
SREFP 3 C00025 BC00025  +REFP EC00025
CALL JOB:SEARCH-R1-S13D
SET P023 P006
SFTON3D P023
SMOVL C00026 BC00026 V=100.0  +MOVJ EC00026
MOVL C00027 BC00027 V=400.0  +MOVJ EC00027 VJ=100.00
SMOVL C00028 BC00028 V=100.0  +MOVJ EC00028
SREFP 3 C00029 BC00029  +REFP EC00029
CALL JOB:SEARCH-R1-S13D
SET P024 P006
SFTON3D P024
SMOVL C00030 BC00030 V=100.0  +MOVJ EC00030
SREFP 3 C00031 BC00031  +REFP EC00031
CALL JOB:SEARCH-R1-S13D
SET P024 P006
SFTON3D P024
SMOVL C00032 BC00032 V=100.0  +MOVJ EC00032
MOVL C00033 BC00033 V=400.0  +MOVJ EC00033 VJ=100.00
MOVL C00034 BC00034 V=1000.0  +MOVJ EC00034 VJ=100.00
'Path S1423
SFTOF3D
SMOVL C00035 BC00035 V=100.0  +MOVJ EC00035
SREFP 3 C00036 BC00036  +REFP EC00036
CALL JOB:SEARCH-R1-S13D
SET P025 P006
SFTON3D P025
SMOVL C00037 BC00037 V=100.0  +MOVJ EC00037
SREFP 3 C00038 BC00038  +REFP EC00038
CALL JOB:SEARCH-R1-S13D
SET P025 P006
SFTON3D P025
SMOVL C00039 BC00039 V=100.0  +MOVJ EC00039
MOVL C00040 BC00040 V=400.0  +MOVJ EC00040 VJ=100.00
MOVL C00041 BC00041 V=1000.0  +MOVJ EC00041 VJ=100.00
'Path S1424
SFTOF3D
SMOVL C00042 BC00042 V=100.0  +MOVJ EC00042
SREFP 3 C00043 BC00043  +REFP EC00043
CALL JOB:SEARCH-R1-S13D
SET P026 P006
SFTON3D P026
SMOVL C00044 BC00044 V=100.0  +MOVJ EC00044
SREFP 3 C00045 BC00045  +REFP EC00045
CALL JOB:SEARCH-R1-S13D
SET P026 P006
SFTON3D P026
SMOVL C00046 BC00046 V=100.0  +MOVJ EC00046
MOVL C00047 BC00047 V=400.0  +MOVJ EC00047 VJ=100.00
MOVJ C00048 BC00048 VJ=50.00  +MOVJ EC00048 VJ=50.00
MOVJ C00049 BC00049 VJ=100.00  +MOVJ EC00049 VJ=50.00
MOVJ C00050 BC00050 VJ=100.00  +MOVJ EC00050 VJ=50.00
MOVJ C00051 BC00051 VJ=100.00  +MOVJ EC00051 VJ=50.00
MOVJ C00052 BC00052 VJ=100.00  +MOVJ EC00052 VJ=50.00
MOVJ C00053 BC00053 VJ=100.00  +MOVJ EC00053 VJ=50.00
SFTOF3D
SMOVL C00054 BC00054 V=166.7  +MOVJ EC00054
SREFP 3 C00055 BC00055  +REFP EC00055
CALL JOB:SEARCH-R1-S13D
SET P027 P006
SFTON3D P027
SMOVL C00056 BC00056 V=100.0  +MOVJ EC00056
SREFP 3 C00057 BC00057  +REFP EC00057
CALL JOB:SEARCH-R1-S13D
SET P027 P006
SFTON3D P027
SMOVL C00058 BC00058 V=100.0  +MOVJ EC00058
SMOVL C00059 BC00059 V=416.7  +MOVJ EC00059
SFTOF3D
SMOVL C00060 BC00060 V=100.0  +MOVJ EC00060
SREFP 3 C00061 BC00061  +REFP EC00061
CALL JOB:SEARCH-R1-S13D
SET P028 P006
SFTON3D P028
SMOVL C00062 BC00062 V=100.0  +MOVJ EC00062
SREFP 3 C00063 BC00063  +REFP EC00063
CALL JOB:SEARCH-R1-S13D
SET P028 P006
SFTON3D P028
SMOVL C00064 BC00064 V=100.0  +MOVJ EC00064
SMOVL C00065 BC00065 V=416.7  +MOVJ EC00065
SMOVL C00066 BC00066 V=416.7  +MOVJ EC00066
SFTOF3D
SMOVL C00067 BC00067 V=100.0  +MOVJ EC00067
SREFP 3 C00068 BC00068  +REFP EC00068
CALL JOB:SEARCH-R1-S13D
SET P029 P006
SFTON3D P029
SMOVL C00069 BC00069 V=100.0  +MOVJ EC00069
SREFP 3 C00070 BC00070  +REFP EC00070
CALL JOB:SEARCH-R1-S13D
SET P029 P006
SFTON3D P029
SMOVL C00071 BC00071 V=100.0  +MOVJ EC00071
MOVJ C00072 BC00072 VJ=100.00  +MOVJ EC00072 VJ=50.00
SFTOF3D
SMOVL C00073 BC00073 V=83.3  +MOVJ EC00073
SREFP 3 C00074 BC00074  +REFP EC00074
CALL JOB:SEARCH-R1-S13D
SET P030 P006
SFTON3D P030
SMOVL C00075 BC00075 V=100.0  +MOVJ EC00075
SREFP 3 C00076 BC00076  +REFP EC00076
CALL JOB:SEARCH-R1-S13D
SET P030 P006
SFTON3D P030
SMOVL C00077 BC00077 V=100.0  +MOVJ EC00077
SFTOF3D
MOVL C00078 BC00078 V=1000.0  +MOVJ EC00078 VJ=100.00
'obrot
MOVJ C00079 BC00079 VJ=100.00  +MOVJ EC00079 VJ=100.00
MOVJ C00080 BC00080 VJ=100.00  +MOVJ EC00080 VJ=100.00
MOVJ C00081 BC00081 VJ=60.00  +MOVJ EC00081 VJ=15.00
MOVJ C00082 BC00082 VJ=100.00  +MOVJ EC00082 VJ=100.00
MOVJ C00083 BC00083 VJ=100.00  +MOVJ EC00083 VJ=100.00
MOVJ C00084 BC00084 VJ=100.00  +MOVJ EC00084 VJ=100.00
MOVJ C00085 BC00085 VJ=100.00  +MOVJ EC00085 VJ=100.00
'Path S1077
SFTOF3D
MOVJ C00086 BC00086 VJ=100.00  +MOVJ EC00086 VJ=100.00
MOVL C00087 BC00087 V=400.0  +MOVJ EC00087 VJ=100.00
SMOVL C00088 BC00088 V=100.0  +MOVJ EC00088
SREFP 3 C00089 BC00089  +REFP EC00089
CALL JOB:SEARCH-R1-S13D
SET P031 P006
SFTON3D P031
SMOVL C00090 BC00090 V=100.0  +MOVJ EC00090
SREFP 3 C00091 BC00091  +REFP EC00091
CALL JOB:SEARCH-R1-S13D
SET P031 P006
SFTON3D P031
SMOVL C00092 BC00092 V=133.3  +MOVJ EC00092
SMOVL C00093 BC00093 V=666.7  +MOVJ EC00093 VJ=100.00
'Path S1078
SFTOF3D
SMOVL C00094 BC00094 V=100.0  +MOVJ EC00094
SREFP 3 C00095 BC00095  +REFP EC00095
CALL JOB:SEARCH-R1-S13D
SET P032 P006
SFTON3D P032
SMOVL C00096 BC00096 V=100.0  +MOVJ EC00096
SREFP 3 C00097 BC00097  +REFP EC00097
CALL JOB:SEARCH-R1-S13D
SET P032 P006
SFTON3D P032
SMOVL C00098 BC00098 V=100.0  +MOVJ EC00098
MOVL C00099 BC00099 V=1000.0  +MOVJ EC00099 VJ=100.00
'Path S1079
SFTOF3D
MOVL C00100 BC00100 V=500.0  +MOVJ EC00100 VJ=100.00
SMOVL C00101 BC00101 V=100.0  +MOVJ EC00101
SREFP 3 C00102 BC00102  +REFP EC00102
CALL JOB:SEARCH-R1-S13D
SET P033 P006
SFTON3D P033
SMOVL C00103 BC00103 V=100.0  +MOVJ EC00103
SREFP 3 C00104 BC00104  +REFP EC00104
CALL JOB:SEARCH-R1-S13D
SET P033 P006
SFTON3D P033
SMOVL C00105 BC00105 V=100.0  +MOVJ EC00105
MOVL C00106 BC00106 V=833.3  +MOVJ EC00106 VJ=100.00
SMOVL C00107 BC00107 V=100.0  +MOVJ EC00107
SREFP 3 C00108 BC00108  +REFP EC00108
CALL JOB:SEARCH-R1-S13D
SET P034 P006
SFTON3D P034
SMOVL C00109 BC00109 V=100.0  +MOVJ EC00109
SREFP 3 C00110 BC00110  +REFP EC00110
CALL JOB:SEARCH-R1-S13D
SET P034 P006
SFTON3D P034
SMOVL C00111 BC00111 V=100.0  +MOVJ EC00111
MOVL C00112 BC00112 V=1000.0  +MOVJ EC00112 VJ=100.00
MOVJ C00113 BC00113 VJ=100.00  +MOVJ EC00113 VJ=50.00
'Path S1078
SFTOF3D
SMOVL C00114 BC00114 V=133.3  +MOVJ EC00114
SREFP 3 C00115 BC00115  +REFP EC00115
CALL JOB:SEARCH-R1-S13D
SET P035 P006
SFTON3D P035
SMOVL C00116 BC00116 V=100.0  +MOVJ EC00116
SREFP 3 C00117 BC00117  +REFP EC00117
CALL JOB:SEARCH-R1-S13D
SET P035 P006
SFTON3D P035
SMOVL C00118 BC00118 V=100.0  +MOVJ EC00118
MOVL C00119 BC00119 V=400.0  +MOVJ EC00119 VJ=100.00
'Path S1079
SFTOF3D
SMOVL C00120 BC00120 V=166.7  +MOVJ EC00120
SREFP 3 C00121 BC00121  +REFP EC00121
CALL JOB:SEARCH-R1-S13D
SET P036 P006
SFTON3D P036
SMOVL C00122 BC00122 V=100.0  +MOVJ EC00122
SREFP 3 C00123 BC00123  +REFP EC00123
CALL JOB:SEARCH-R1-S13D
SET P036 P006
SFTON3D P036
SMOVL C00124 BC00124 V=100.0  +MOVJ EC00124
SFTOF3D
MOVJ C00125 BC00125 VJ=100.00  +MOVJ EC00125 VJ=50.00
MOVJ C00126 BC00126 VJ=100.00  +MOVJ EC00126 VJ=50.00
MOVJ C00127 BC00127 VJ=100.00  +MOVJ EC00127 VJ=50.00
MOVJ C00128 BC00128 VJ=100.00  +MOVJ EC00128 VJ=50.00
MOVJ C00129 BC00129 VJ=100.00  +MOVJ EC00129 VJ=50.00
MOVJ C00130 BC00130 VJ=100.00  +MOVJ EC00130 VJ=50.00
SMOVL C00131 BC00131 V=100.0  +MOVJ EC00131
SREFP 3 C00132 BC00132  +REFP EC00132
CALL JOB:SEARCH-R1-S13D
SET P037 P006
SFTON3D P037
SMOVL C00133 BC00133 V=100.0  +MOVJ EC00133
SREFP 3 C00134 BC00134  +REFP EC00134
CALL JOB:SEARCH-R1-S13D
SET P037 P006
SFTON3D P037
SMOVL C00135 BC00135 V=100.0  +MOVJ EC00135
MOVL C00136 BC00136 V=333.3  +MOVJ EC00136 VJ=100.00
'Path S1078
SFTOF3D
SMOVL C00137 BC00137 V=100.0  +MOVJ EC00137
SREFP 3 C00138 BC00138  +REFP EC00138
CALL JOB:SEARCH-R1-S13D
SET P038 P006
SFTON3D P038
SMOVL C00139 BC00139 V=100.0  +MOVJ EC00139
SREFP 3 C00140 BC00140  +REFP EC00140
CALL JOB:SEARCH-R1-S13D
SET P038 P006
SFTON3D P038
SMOVL C00141 BC00141 V=100.0  +MOVJ EC00141
MOVL C00142 BC00142 V=333.3  +MOVJ EC00142 VJ=100.00
'Path S1079
SFTOF3D
MOVL C00143 BC00143 V=400.0  +MOVJ EC00143 VJ=100.00
MOVJ C00144 BC00144 VJ=100.00  +MOVJ EC00144 VJ=50.00
SMOVL C00145 BC00145 V=133.3  +MOVJ EC00145
SREFP 3 C00146 BC00146  +REFP EC00146
CALL JOB:SEARCH-R1-S13D
SET P039 P006
SFTON3D P039
SMOVL C00147 BC00147 V=100.0  +MOVJ EC00147
SREFP 3 C00148 BC00148  +REFP EC00148
CALL JOB:SEARCH-R1-S13D
SET P039 P006
SFTON3D P039
SMOVL C00149 BC00149 V=166.7  +MOVJ EC00149
SFTON3D P039
SMOVL C00150 BC00150 V=166.7 PL=0  +MOVJ EC00150
SREFP 1 C00151 BC00151  +REFP EC00151
SREFP 2 C00152 BC00152  +REFP EC00152
MACRO1 MJ#(0) ARGF14
ARCON
SMOVL C00153 BC00153 V=10.0  +MOVJ EC00153
ARCOF
SFTOF3D
SMOVL C00154 BC00154 V=166.7  +MOVJ EC00154
SMOVL C00155 BC00155 V=416.7  +MOVJ EC00155
SFTOF3D
SFTON3D P037
SMOVL C00156 BC00156 V=133.3 PL=0  +MOVJ EC00156
SREFP 1 C00157 BC00157  +REFP EC00157
SREFP 2 C00158 BC00158  +REFP EC00158
MACRO1 MJ#(0) ARGF17
ARCON
SFTON3D P038
SMOVL C00159 BC00159 V=11.2  +MOVJ EC00159
ARCOF
SFTOF3D
SMOVL C00160 BC00160 V=400.0  +MOVJ EC00160
SMOVL C00161 BC00161 V=250.0  +MOVJ EC00161
MOVJ C00162 BC00162 VJ=100.00  +MOVJ EC00162 VJ=100.00
MOVJ C00163 BC00163 VJ=100.00  +MOVJ EC00163 VJ=100.00
MOVJ C00164 BC00164 VJ=60.00  +MOVJ EC00164 VJ=60.00
MOVJ C00165 BC00165 VJ=60.00  +MOVJ EC00165 VJ=60.00
MOVJ C00166 BC00166 VJ=60.00  +MOVJ EC00166 VJ=60.00
MOVJ C00167 BC00167 VJ=100.00  +MOVJ EC00167 VJ=100.00
MOVJ C00168 BC00168 VJ=100.00  +MOVJ EC00168 VJ=100.00
MOVJ C00169 BC00169 VJ=100.00  +MOVJ EC00169 VJ=100.00
SMOVL C00170 BC00170 V=1000.0  +MOVJ EC00170
SFTOF3D
SFTON3D P032
SMOVL C00171 BC00171 V=133.3 PL=0  +MOVJ EC00171
SREFP 1 C00172 BC00172  +REFP EC00172
SREFP 2 C00173 BC00173  +REFP EC00173
MACRO1 MJ#(0) ARGF14
ARCON
SMOVL C00174 BC00174 V=10.0  +MOVJ EC00174
ARCOF
SMOVL C00175 BC00175 V=400.0  +MOVJ EC00175
SMOVL C00176 BC00176 V=333.3  +MOVJ EC00176
SFTON3D P031
SMOVL C00177 BC00177 V=133.3 PL=0  +MOVJ EC00177
SREFP 1 C00178 BC00178  +REFP EC00178
SREFP 2 C00179 BC00179  +REFP EC00179
MACRO1 MJ#(0) ARGF14
ARCON
SMOVL C00180 BC00180 V=10.0  +MOVJ EC00180
ARCOF
SMOVL C00181 BC00181 V=400.0  +MOVJ EC00181
SMOVL C00182 BC00182 V=250.0  +MOVJ EC00182
SFTON3D P034
SMOVL C00183 BC00183 V=133.3 PL=0  +MOVJ EC00183
SREFP 1 C00184 BC00184  +REFP EC00184
SREFP 2 C00185 BC00185  +REFP EC00185
MACRO1 MJ#(0) ARGF14
ARCON
SMOVL C00186 BC00186 V=10.0  +MOVJ EC00186
ARCOF
SMOVL C00187 BC00187 V=400.0  +MOVJ EC00187
SMOVL C00188 BC00188 V=666.7  +MOVJ EC00188
SFTON3D P033
SMOVL C00189 BC00189 V=133.3 PL=0  +MOVJ EC00189
SREFP 1 C00190 BC00190  +REFP EC00190
SREFP 2 C00191 BC00191  +REFP EC00191
MACRO1 MJ#(0) ARGF14
ARCON
SMOVL C00192 BC00192 V=10.0  +MOVJ EC00192
ARCOF
SMOVL C00193 BC00193 V=1000.0  +MOVJ EC00193
SMOVL C00194 BC00194 V=500.0  +MOVJ EC00194
SFTON3D P036
SMOVL C00195 BC00195 V=133.3 PL=0  +MOVJ EC00195
SREFP 1 C00196 BC00196  +REFP EC00196
SREFP 2 C00197 BC00197  +REFP EC00197
MACRO1 MJ#(0) ARGF14
ARCON
SMOVL C00198 BC00198 V=10.0  +MOVJ EC00198
ARCOF
SMOVL C00199 BC00199 V=400.0  +MOVJ EC00199
SMOVL C00200 BC00200 V=500.0  +MOVJ EC00200
'SPRAWDZIC SPOINE
SFTON3D P035
SMOVL C00201 BC00201 V=133.3 PL=0  +MOVJ EC00201
SREFP 1 C00202 BC00202  +REFP EC00202
SREFP 2 C00203 BC00203  +REFP EC00203
MACRO1 MJ#(0) ARGF14
ARCON
SMOVL C00204 BC00204 V=10.0  +MOVJ EC00204
ARCOF
SMOVL C00205 BC00205 V=666.7  +MOVJ EC00205
MOVJ C00206 BC00206 VJ=100.00  +MOVJ EC00206 VJ=50.00
'obrot
MOVJ C00207 BC00207 VJ=100.00  +MOVJ EC00207 VJ=100.00
MOVJ C00208 BC00208 VJ=100.00  +MOVJ EC00208 VJ=100.00
MOVJ C00209 BC00209 VJ=100.00  +MOVJ EC00209 VJ=100.00
MOVJ C00210 BC00210 VJ=100.00  +MOVJ EC00210 VJ=100.00
MOVJ C00211 BC00211 VJ=100.00  +MOVJ EC00211 VJ=100.00
MOVJ C00212 BC00212 VJ=100.00  +MOVJ EC00212 VJ=100.00
MOVJ C00213 BC00213 VJ=100.00  +MOVJ EC00213 VJ=100.00
'Path W1425
SFTOF3D
SFTON3D P023
MOVJ C00214 BC00214 VJ=100.00  +MOVJ EC00214 VJ=100.00
SMOVL C00215 BC00215 V=333.3  +MOVJ EC00215
SMOVL C00216 BC00216 V=133.3 PL=0  +MOVJ EC00216
SREFP 1 C00217 BC00217  +REFP EC00217
SREFP 2 C00218 BC00218  +REFP EC00218
MACRO1 MJ#(0) ARGF14
ARCON
SMOVL C00219 BC00219 V=10.0  +MOVJ EC00219
ARCOF
SMOVL C00220 BC00220 V=400.0  +MOVJ EC00220
SMOVL C00221 BC00221 V=1000.0  +MOVJ EC00221
SFTOF3D
SFTON3D P022
MOVJ C00222 BC00222 VJ=100.00  +MOVJ EC00222 VJ=100.00
SMOVL C00223 BC00223 V=133.3 PL=0  +MOVJ EC00223
SREFP 1 C00224 BC00224  +REFP EC00224
SREFP 2 C00225 BC00225  +REFP EC00225
MACRO1 MJ#(0) ARGF14
ARCON
SMOVL C00226 BC00226 V=10.0  +MOVJ EC00226
ARCOF
SMOVL C00227 BC00227 V=400.0  +MOVJ EC00227
SMOVL C00228 BC00228 V=1000.0  +MOVJ EC00228
SFTOF3D
SFTON3D P021
MOVJ C00229 BC00229 VJ=100.00  +MOVJ EC00229 VJ=100.00
SMOVL C00230 BC00230 V=133.3 PL=0  +MOVJ EC00230
SREFP 1 C00231 BC00231  +REFP EC00231
SREFP 2 C00232 BC00232  +REFP EC00232
MACRO1 MJ#(0) ARGF14
ARCON
SMOVL C00233 BC00233 V=10.0  +MOVJ EC00233
ARCOF
SMOVL C00234 BC00234 V=400.0  +MOVJ EC00234
SMOVL C00235 BC00235 V=333.3  +MOVJ EC00235
SFTON3D P026
SMOVL C00236 BC00236 V=133.3 PL=0  +MOVJ EC00236
SREFP 1 C00237 BC00237  +REFP EC00237
SREFP 2 C00238 BC00238  +REFP EC00238
MACRO1 MJ#(0) ARGF14
ARCON
SMOVL C00239 BC00239 V=10.0  +MOVJ EC00239
ARCOF
SMOVL C00240 BC00240 V=400.0  +MOVJ EC00240
SMOVL C00241 BC00241 V=1000.0  +MOVJ EC00241
SFTOF3D
SFTON3D P025
SMOVL C00242 BC00242 V=133.3 PL=0  +MOVJ EC00242
SREFP 1 C00243 BC00243  +REFP EC00243
SREFP 2 C00244 BC00244  +REFP EC00244
MACRO1 MJ#(0) ARGF14
ARCON
SMOVL C00245 BC00245 V=10.0  +MOVJ EC00245
ARCOF
SMOVL C00246 BC00246 V=400.0  +MOVJ EC00246
SMOVL C00247 BC00247 V=1000.0  +MOVJ EC00247
SFTOF3D
'Path W1427
SFTOF3D
SFTON3D P024
SMOVL C00248 BC00248 V=133.3 PL=0  +MOVJ EC00248
SREFP 1 C00249 BC00249  +REFP EC00249
SREFP 2 C00250 BC00250  +REFP EC00250
MACRO1 MJ#(0) ARGF14
ARCON
SMOVL C00251 BC00251 V=10.0  +MOVJ EC00251
ARCOF
SMOVL C00252 BC00252 V=400.0  +MOVJ EC00252
MOVJ C00253 BC00253 VJ=100.00  +MOVJ EC00253 VJ=100.00
MOVJ C00254 BC00254 VJ=100.00  +MOVJ EC00254 VJ=100.00
MOVJ C00255 BC00255 VJ=100.00  +MOVJ EC00255 VJ=100.00
MOVJ C00256 BC00256 VJ=100.00  +MOVJ EC00256 VJ=100.00
MOVJ C00257 BC00257 VJ=100.00  +MOVJ EC00257 VJ=100.00
MOVJ C00258 BC00258 VJ=100.00  +MOVJ EC00258 VJ=100.00
SFTON3D P027
SMOVL C00259 BC00259 V=166.7  +MOVJ EC00259
ARCON
SMOVL C00260 BC00260 V=10.0  +MOVJ EC00260
ARCOF
SFTOF3D
MOVJ C00261 BC00261 VJ=100.00  +MOVJ EC00261 VJ=100.00
MOVJ C00262 BC00262 VJ=100.00  +MOVJ EC00262 VJ=100.00
MOVJ C00263 BC00263 VJ=100.00  +MOVJ EC00263 VJ=100.00
SFTON3D P030
SMOVL C00264 BC00264 V=133.3  +MOVJ EC00264
ARCON
SFTON3D P029
SMOVL C00265 BC00265 V=10.0  +MOVJ EC00265
ARCOF
SFTOF3D
SMOVL C00266 BC00266 V=250.0  +MOVJ EC00266
MOVJ C00267 BC00267 VJ=100.00  +MOVJ EC00267 VJ=100.00
MOVJ C00268 BC00268 VJ=100.00  +MOVJ EC00268 VJ=100.00
MOVJ C00269 BC00269 VJ=100.00  +MOVJ EC00269 VJ=100.00
'KONIEC
END
